// Mitsubishi GX Works2 project: and_3i_nputs   PLC: Q03UDV
// LRI_2023

PROGRAM MAIN
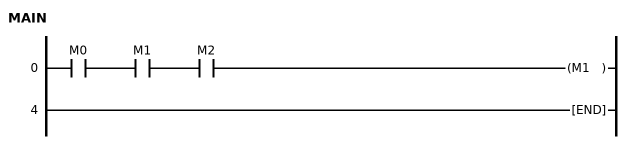
0     LD      M0
      AND     M1
      AND     M2
      OUT     M1
4     END
END_PROGRAM
